TEXTLIST TextList
  1 = 'Profile Position'
  3 = 'Profile Velocity'
  4 = 'Profile Torque'
  8 = 'Cyclic Sync Position'
  9 = 'Cyclic Sync Velocity'
  10 = 'Cyclic Sync Torque'
   = ''
END_TEXTLIST

(* stored: Version 1.1.0.1, ProductVersion 3.1.4024.11
   TextList TextList: Id {ab44bbef-7e42-4df1-8fce-f12877b21bd9} *)
